FUNCTION IsErr : BOOL
VAR_INPUT
	eResult			: Result;
END_VAR
VAR_OUTPUT
	eCarry			: Result;
END_VAR

IsErr := eResult < 0;
eCarry := eResult;

END_FUNCTION

(* stored: Version 1.1.0.1
   POU IsErr: Id {d8e5ecc7-39a3-4a90-b2be-f8d0e55647cb}, SpecialFunc None *)
